{attribute 'reflection'} 
FUNCTION_BLOCK FB_Testsuite EXTENDS FB_Base IMPLEMENTS I_Testsuite
VAR_INPUT
END_VAR
VAR_OUTPUT
END_VAR
VAR
	iParent:			I_Testsuites;
	fCycleTime: 		LREAL;	
	stTestsuite:		ST_Testsuite;
	stTestcase:			ST_Testcase;
	fbBuilder:			FB_StringBuilder;
	fbList:				FB_ListSTRING;
	fbAssert:			FB_Assert;
	nActual:			INT:=  E_Testcase.Init;
	nNext:				INT;
	fbTimeout:			TON;
END_VAR

SUPER^();

METHOD PROTECTED M_Started : BOOL
VAR_INPUT
END_VAR
VAR
	nIndex: DINT;
	sValue: STRING(255);
END_VAR
stTestcase.nAssertions:= fbAssert.nAssert;
IF fbAssert.nPassed = fbAssert.nAssert THEN
	fbBuilder.M_Reset();
	fbBuilder.M_Append('<testcase name="');
	fbBuilder.M_Append(stTestCase.sName);
	fbBuilder.M_Append('" classname="');
	fbBuilder.M_Append(stTestCase.sClassname);
	fbBuilder.M_Append('" assertions="');
	fbBuilder.M_AppendInt(stTestCase.nAssertions);
	fbBuilder.M_Append('" time="');
	fbBuilder.M_AppendReal(stTestCase.fTime, 5);
	fbBuilder.M_Append('" file="');
	fbBuilder.M_Append(stTestCase.sFile);
	fbBuilder.M_Append('" line="');
	fbBuilder.M_AppendInt(stTestCase.nLine);
	fbBuilder.M_Append('" />');
	fbBuilder.M_Copy(sValue);
	fbList.M_Add(sValue);

	stTestsuite.nTests:= stTestsuite.nTests + 1;
	stTestsuite.nFailures:= stTestsuite.nFailures + fbAssert.nFailures;
	stTestsuite.nErrors:= stTestsuite.nErrors + fbAssert.nErrors;
	stTestsuite.nSkipped:= stTestsuite.nSkipped + fbAssert.nSkipped;
	stTestsuite.nAssertions:= stTestsuite.nAssertions + fbAssert.nAssert;
	stTestsuite.fTime:= stTestsuite.fTime + stTestCase.fTime;
	stTestCase.fTime:= -fCycleTime;
	fbTimeout(IN:=FALSE);
	nActual:= nNext;
ELSE
	IF fbTimeout.Q THEN
		fbBuilder.M_Reset();
		fbBuilder.M_Append('<testcase name="');
		fbBuilder.M_Append(stTestCase.sName);
		fbBuilder.M_Append('" classname="');
		fbBuilder.M_Append(stTestCase.sClassname);
		fbBuilder.M_Append('" assertions="');
		fbBuilder.M_AppendInt(stTestCase.nAssertions);
		fbBuilder.M_Append('" time="');
		fbBuilder.M_AppendReal(stTestCase.fTime, 5);
		fbBuilder.M_Append('" file="');
		fbBuilder.M_Append(stTestCase.sFile);
		fbBuilder.M_Append('" line="');
		fbBuilder.M_AppendInt(stTestCase.nLine);
		fbBuilder.M_Append('" >');
		WHILE nIndex < fbAssert.fbList.P_Length DO
			fbBuilder.M_Append(fbAssert.fbList.M_Item(nIndex));
			nIndex:= nIndex + 1;
		END_WHILE
		fbBuilder.M_Append('</testcase>');
		fbBuilder.M_Copy(sValue);
		fbList.M_Add(sValue);
		stTestsuite.nTests:= stTestsuite.nTests + 1;
		stTestsuite.nFailures:= stTestsuite.nFailures + fbAssert.nFailures;
		stTestsuite.nErrors:= stTestsuite.nErrors + fbAssert.nErrors;
		stTestsuite.nSkipped:= stTestsuite.nSkipped + fbAssert.nSkipped;
		stTestsuite.nAssertions:= stTestsuite.nAssertions + fbAssert.nAssert;
		stTestsuite.fTime:= stTestsuite.fTime + stTestCase.fTime;
		stTestCase.fTime:= -fCycleTime;
		fbTimeout(IN:=FALSE);
		nActual:= nNext;
	END_IF
END_IF
stTestcase.fTime:= stTestcase.fTime + fCycleTime;
fbAssert.M_Reset();
M_Started:= nActual = E_Testcase.Done;
END_METHOD

METHOD PROTECTED M_Starting : BOOL
VAR_INPUT
END_VAR

VAR
	nIndex: DINT;
END_VAR
CASE nState OF
	0:
		IF 	SUPER^.M_Starting() THEN
			fbList.M_Clear();
			fCycleTime:= F_GetCycleTime();	
			stTestsuite.sName:= F_GetName(sInstancePath);
			stTestsuite.nTests:= 0;
			stTestsuite.nFailures:= 0;		
			stTestsuite.nErrors:= 0;	
			stTestsuite.nSkipped:= 0;		
			stTestsuite.nAssertions:= 0;	
			stTestsuite.fTime:= 0.0;
			stTestsuite.sFile:= '';
			nState:= 1;
		END_IF
		
	1:
		nActual:= E_Testcase.Start;
		M_Starting:= TRUE;
	
END_CASE
END_METHOD

METHOD PROTECTED M_Stopping : BOOL
VAR_INPUT
END_VAR
VAR
	sValue: STRING(255);
	nIndex: DINT;
END_VAR
//    <testsuite name="Tests.Registration" tests="8" failures="1" errors="1" skipped="1" assertions="20" time="16.082687" timestamp="2021-04-02T15:48:23" file="tests/registration.code">
fbBuilder.M_Reset();
fbBuilder.M_Append('<testsuite name="');
fbBuilder.M_Append(stTestsuite.sName);
fbBuilder.M_Append('" tests="');
fbBuilder.M_AppendInt(stTestsuite.nTests);
fbBuilder.M_Append('" failures="');
fbBuilder.M_AppendInt(stTestsuite.nFailures);
fbBuilder.M_Append('" errors="');
fbBuilder.M_AppendInt(stTestsuite.nErrors);
fbBuilder.M_Append('" skipped="');
fbBuilder.M_AppendInt(stTestsuite.nSkipped);
fbBuilder.M_Append('" assertions="');
fbBuilder.M_AppendInt(stTestsuite.nAssertions);	
fbBuilder.M_Append('" time="');
fbBuilder.M_AppendReal(stTestsuite.fTime, 4);
fbBuilder.M_Append('" timestamp="');
fbBuilder.M_Append(stTestsuite.sTimestamp);
fbBuilder.M_Append('" file="');
fbBuilder.M_Append(stTestsuite.sFile);
fbBuilder.M_Append('">');
fbBuilder.M_Copy(sValue);
fbList.M_Insert(0, sValue);
fbList.M_Add('</testsuite>');
IF iParent <> 0 THEN
	WHILE nIndex < fbList.P_Length DO
		iParent.P_List.M_Add(fbList.M_Item(nIndex));
	END_WHILE
END_IF
M_Stopping:= TRUE;
END_METHOD

METHOD PUBLIC M_Testcase : BOOL
VAR_INPUT
	Classname:			STRING(255);	// Classname as string
	Timeout:			TIME;			// Timeout in ms
	File:				STRING(255);
	Line:				DINT;	
	Next:				INT;			// Next test case
END_VAR
stTestcase.sName:= CONCAT(CONCAT(CONCAT(stTestsuite.sName,'.'), 'M_Testcase-'), INT_TO_STRING(nActual));
stTestcase.sClassname:= Classname;
stTestcase.nAssertions:= fbAssert.fbList.P_Length;
stTestcase.sFile:= File;
stTestcase.NLine:= Line;
IF Timeout <> T#0S THEN
	fbTimeout(IN:= TRUE, PT:= Timeout);
END_IF
nNext:= Next;
END_METHOD

PROPERTY PUBLIC P_Assert : I_Assert
GET
P_Assert:= fbAssert;
END_GET
END_PROPERTY

PROPERTY PUBLIC P_List : I_ListSTRING
GET
P_List:= fbList;
END_GET
END_PROPERTY

PROPERTY PUBLIC P_Parent : I_Testsuites
GET
P_Parent:= iParent;
END_GET
SET
iParent:= P_Parent;
END_SET
END_PROPERTY

PROPERTY PUBLIC P_Result : ST_Testsuite
GET
P_Result:= stTestsuite;
END_GET
END_PROPERTY

PROPERTY PUBLIC P_Testcase : int
GET
P_Testcase:= nActual;
END_GET
END_PROPERTY

END_FUNCTION_BLOCK

(* stored: Version 1.1.0.1
   POU FB_Testsuite: Id {139d3d86-4160-0b84-0f97-b2398a2924e9}, SpecialFunc None
   Method M_Started: Id {78e3f5cf-1c2d-00e7-2cad-335430cad839}
   Method M_Starting: Id {fa2aca87-7276-0f36-03ec-8cf918759ac1}
   Method M_Stopping: Id {86997241-28ad-050a-3199-6300c2ef6b3b}
   Method M_Testcase: Id {6d08bc5e-dc98-0f10-1d34-7f069e37b9d3}
   Property P_Assert: Id {e23dc60a-455c-05e0-203b-c87d7f0bf2be}
   Get Get: Id {af1ab888-05f6-09a5-0125-87c54b409f9b}
   Property P_List: Id {37feeb7c-033b-03ab-2f25-c1e23d6d59c4}
   Get Get: Id {00de385f-f60f-01e8-2c65-d740b8aed217}
   Property P_Parent: Id {26b3c1be-b48f-0a73-3f11-669666d67824}
   Get Get: Id {cbeb0dff-5be2-0eeb-3c4b-d2308bd2f226}
   Set Set: Id {b6a9fa31-34bd-0c5b-2292-21f39b156b39}
   Property P_Result: Id {bc6fd8b0-043c-05d2-0765-58761c6f620a}
   Get Get: Id {3423e8a5-6264-06ea-335d-82063928e5f1}
   Property P_Testcase: Id {3b7b6a2e-6d4a-0f0e-2a1d-3d960844879b}
   Get Get: Id {854def52-87cb-03f8-22d6-ee5144597bf5} *)
